{attribute 'qualified_only'}
{attribute 'strict'}
TYPE
    eCUState :
    (
        None       := 0,
        HasWarning := 10,
        HasError   := 20
    );
END_TYPE

(* stored: Version 1.1.0.1
   DUT eCUState: Id {9a45f02b-5396-0221-3c94-d40625fb654b} *)
